// TwinCAT 3 PLC project Untitled1
// ProgramVersion: 3.1.4023.0
// libraries:
//   Tc2_Standard, * (Beckhoff Automation GmbH)
//   Tc2_System, * (Beckhoff Automation GmbH)
//   Tc3_Module, * (Beckhoff Automation GmbH)
// project tree:
//   / PlcTask.TcTTO (not stored)
//   POUs/ MAIN.TcPOU
// real-time tasks:
//   TASK PlcTask: cycle T#10ms, priority 20, ADS port 350
// I/O:
//   DEVICE EtherCAT_Master_EJxxxx, AmsNetId 172.20.30.238.7.1
//     Beckhoff EJ1xxx [EK1100 EtherCAT Coupler (2A E-Bus)]
//       Beckhoff EJ1xxxEK1122 [EK1122 2 port EtherCAT junction]
//         Beckhoff EJ1xxxsub EK1100 [EK1100 EtherCAT Coupler (2A E-Bus)]
//         A_0001(EJ1100-0000-0018) [EJ1100 EtherCAT Coupler (2.2A E-Bus)]
//         A_0002(EJ1101-0022-0016) [EJ1101-0022 EtherCAT Coupler (ID switch)]
//       A_0004(EJ1008-0000-0017) [EJ1008 8Ch. Dig. Input 24V, 3ms]
//       A_0005(EJ1128-0000-0016) [EJ1128 8Ch. Dig. Input 5V / 3.3V DC, 0.05µs]
//       A_0006(EJ1809-0000-0017) [EJ1809 16Ch. Dig. Input 24V, 3ms]
//       A_0007(EJ1819-0000-0017) [EJ1819 16Ch. Dig. Input 24V, 10µs]
//       A_0008(EJ1859-0000-0017) [EJ1859 8Ch. Dig. Input 24V, 3ms, 8Ch. Dig. Output 24V, 0.5A]
//       A_0009(EJ1889-0000-0017) [EJ1889 16Ch. Dig. Input 24V, 3ms, negative]
//       A_0003(EJ1122-0000-0016) [EJ1122 2 port EtherCAT junction]
//     Beckhoff EJ2xxx [EK1100 EtherCAT Coupler (2A E-Bus)]
//       Beckhoff EJ2xxxEK1122 [EK1122 2 port EtherCAT junction]
//         Beckhoff EJ2xxxsub EK1100 [EK1100 EtherCAT Coupler (2A E-Bus)]
//       A_0001(EJ2008-0000-0017) [EJ2008 8Ch. Dig. Output 24V, 0.5A]
//       A_0002(EJ2008-0000-0018) [EJ2008 8Ch. Dig. Output 24V, 0.5A]
//       A_0003(EJ2128-0000-0016) [EJ2128 8Ch. Dig. Output 5V/3.3V, 20mA]
//       A_0004(EJ2502-0000-0023) [EJ2502 2Ch. PWM output, 24V]
//       A_0005(EJ2502-0000-0024) [EJ2502 2Ch. PWM output, 24V]
//       A_0006(EJ2521-0224-0016) [EJ2521-0224 1Ch. Pulse Train 24V DC Output Capture/Compare]
//       A_0007(EJ2522-0000-0022) [EJ2522 2Ch. Pulse Train Output]
//       A_0008(EJ2809-0000-0017) [EJ2809 16Ch. Dig. Output 24V, 0.5A]
//       A_0009(EJ2889-0000-0016) [EJ2889 16Ch. Dig. Output 24V, 0.5A, negative]
//       A_0010(EJ2889-0000-0017) [EJ2889 16Ch. Dig. Output 24V, 0.5A, negative]
//     Beckhoff EJ3xxx [EK1100 EtherCAT Coupler (2A E-Bus)]
//       Beckhoff EJ3xxxEK1122 [EK1122 2 port EtherCAT junction]
//         Beckhoff EJ3xxxsub EK1100 [EK1100 EtherCAT Coupler (2A E-Bus)]
//       A_0001(EJ3004-0000-0019) [EJ3004 4Ch. Ana. Input +/-10V]
//       A_0002(EJ3004-0000-0020) [EJ3004 4Ch. Ana. Input +/-10V]
//       A_0003(EJ3004-0000-0021) [EJ3004 4Ch. Ana. Input +/-10V]
//       A_0004(EJ3048-0000-0020) [EJ3048 8Ch. Ana. Input 0-20mA]
//       A_0005(EJ3058-0000-0020) [EJ3058 8Ch. Ana. Input 4-20mA]
//       A_0006(EJ3068-0000-0020) [EJ3068 8Ch. Ana. Input 0-10V]
//       A_0007(EJ3068-0000-0021) [EJ3068 8Ch. Ana. Input 0-10V]
//       A_0008(EJ3104-0000-0019) [EJ3104 4Ch. Ana. Input +/-10V DIFF]
//       A_0009(EJ3104-0000-0020) [EJ3104 4Ch. Ana. Input +/-10V DIFF]
//       A_0010(EJ3104-0000-0021) [EJ3104 4Ch. Ana. Input +/-10V DIFF]
//       A_0011(EJ3108-0000-0017) [EJ3108 8Ch. Ana. Input +/-10V]
//       A_0012(EJ3108-0000-0018) [EJ3108 8Ch. Ana. Input +/-10V]
//       A_0013(EJ3108-0000-0019) [EJ3108 8Ch. Ana. Input +/-10V]
//       A_0014(EJ3202-0000-0019) [EJ3202 2Ch. Ana. Input PT100 (RTD)]
//       A_0015(EJ3202-0000-0020) [EJ3202 2Ch. Ana. Input PT100 (RTD)]
//       A_0016(EJ3202-0000-0021) [EJ3202 2Ch. Ana. Input PT100 (RTD)]
//       A_0017(EJ3214-0000-0016) [EJ3214 4Ch. Ana. Input PT100 (RTD)]
//       A_0018(EJ3255-0000-0023) [EJ3255 5Ch. potentiometer measurement with sensor supply]
//       A_0019(EJ3318-0000-0017) [EJ3318 8Ch. Ana Input Thermocouple (TC)]
//     Beckhoff EJ4xxx [EK1100 EtherCAT Coupler (2A E-Bus)]
//       Beckhoff EJ4xxxEK1122 [EK1122 2 port EtherCAT junction]
//         Beckhoff EJ4xxxsub EK1100 [EK1100 EtherCAT Coupler (2A E-Bus)]
//       A_0001(EJ4002-0000-0017) [EJ4002 2Ch. Ana. Output 0-10V, 12bit]
//       A_0002(EJ4002-0000-0018) [EJ4002 2Ch. Ana. Output 0-10V, 12bit]
//       A_0003(EJ4004-0000-0020) [EJ4004 4Ch. Ana. Output 0-10V, 12bit]
//       A_0004(EJ4008-0000-0020) [EJ4008 8Ch. Ana. Output 0-10V, 12bit]
//       A_0005(EJ4018-0000-0016) [EJ4018 8Ch. Ana. Output 0-20mA, 12bit]
//       A_0006(EJ4024-0000-0020) [EJ4024 4Ch. Ana. Output 4-20mA, 12bit]
//       A_0007(EJ4132-0000-0019) [EJ4132 2Ch. Ana. Output -10/+10V, 16bit]
//       A_0008(EJ4134-0000-0019) [EJ4134 4Ch. Ana. Output -10/+10V, 16bit]
//       A_0009(EJ4134-0000-0020) [EJ4134 4Ch. Ana. Output -10/+10V, 16bit]
//     Beckhoff EJ5xxx [EK1100 EtherCAT Coupler (2A E-Bus)]
//       Beckhoff EJ5xxxEK1122 [EK1122 2 port EtherCAT junction]
//         Beckhoff EJ5xxxsub EK1100 [EK1100 EtherCAT Coupler (2A E-Bus)]
//       A_0001(EJ5002-0000-0016) [EJ5002 2Ch. SSI Encoder]
//       A_0002(EJ5002-0000-0017) [EJ5002 2Ch. SSI Encoder]
//       A_0003(EJ5101-0000-0016) [EJ5101 1Ch. Inc. Encoder 5V]
//       A_0004(EJ5151-0000-0016) [EJ5151 1Ch. Inc. Encoder]
//     Beckhoff EJ6xxx [EK1100 EtherCAT Coupler (2A E-Bus)]
//       Beckhoff EJ6xxxEK1122 [EK1122 2 port EtherCAT junction]
//         Beckhoff EJ6xxxsub EK1100 [EK1100 EtherCAT Coupler (2A E-Bus)]
//       A_0001(EJ6002-0000-0016) [EJ6002 Interface 2Ch. (RS232/RS485/RS422)]
//       A_0002(EJ6224-0000-0016) [EJ6224 (IO Link Master)]
//         modules: Module 1 (DeviceState Inputs Device), Module 2 (DeviceState Inputs), Module 3 (empty), Module 4 (empty), Module 5 (empty), Module 6 (empty)
//       A_0003(EJ6224-0090-0016) [EJ6224-0090 (IO Link Master, TwinSAFE SC)]
//         modules: Module 1 (DeviceState Inputs Device), Module 2 (DeviceState Inputs), Module 3 (empty), Module 4 (empty), Module 5 (empty), Module 6 (empty)
//     Beckhoff EJ7xxx [EK1100 EtherCAT Coupler (2A E-Bus)]
//       Beckhoff EJ7xxxEK1122 [EK1122 2 port EtherCAT junction]
//         Beckhoff EJ7xxxsub EK1100 [EK1100 EtherCAT Coupler (2A E-Bus)]
//       A_0001(EJ7031-0000-0026) [EJ7031 1Ch. Stepper motor output stage (24V, 1.5A)]
//       A_0002(EJ7037-0000-0020) [EJ7037 1Ch. Stepper motor output stage (24V, 1.5A)]
//       A_0003(EJ7041-0052-0016) [EJ7041-0052 1Ch. Stepper motor output stage (50V, 5A)]
//       A_0004(EJ7047-0000-0018) [EJ7047 1Ch. Stepper motor output stage (50V, 5A)]
//       A_0005(EJ7047-0000-0019) [EJ7047 1Ch. Stepper motor output stage (50V, 5A)]
//       A_0006(EJ7047-0000-0020) [EJ7047 1Ch. Stepper motor output stage (50V, 5A)]
//       A_0007(EJ7342-0000-0019) [EJ7342 2Ch. DC motor output stage (50V, 3.5A)]
//       A_0008(EJ7342-0000-0020) [EJ7342 2Ch. DC motor output stage (50V, 3.5A)]
//       A_0009(EJ7211-0010-0026) [EJ7211-0010 1Ch. MDP742 Servo motor output stage with OCT (50V, 4.5A RMS)]
//       A_0010(EJ7211-0010-0027) [EJ7211-0010 1Ch. MDP742 Servo motor output stage with OCT (50V, 4.5A RMS)]
//       A_0011(EJ7211-0010-0028) [EJ7211-0010 1Ch. MDP742 Servo motor output stage with OCT (50V, 4.5A RMS)]
//       A_0012(EJ7211-0010-0029) [EJ7211-0010 1Ch. MDP742 Servo motor output stage with OCT (50V, 4.5A RMS)]
//       A_0013(EJ7211-0010-0030) [EJ7211-0010 1Ch. MDP742 Servo motor output stage with OCT (50V, 4.5A RMS)]
//       A_0014(EJ7211-0010-0031) [EJ7211-0010 1Ch. MDP742 Servo motor output stage with OCT (50V, 4.5A RMS)]
//       A_0015(EJ7211-0010-0032) [EJ7211-0010 1Ch. MDP742 Servo motor output stage with OCT (50V, 4.5A RMS)]
//       A_0016(EJ7211-0011-0026) [EJ7211-0011 1Ch. DS402 Servo motor output stage with OCT (50V, 4.5A RMS)]
//       A_0017(EJ7211-0011-0027) [EJ7211-0011 1Ch. DS402 Servo motor output stage with OCT (50V, 4.5A RMS)]
//       A_0018(EJ7211-0011-0028) [EJ7211-0011 1Ch. DS402 Servo motor output stage with OCT (50V, 4.5A RMS)]
//       A_0019(EJ7211-0011-0029) [EJ7211-0011 1Ch. DS402 Servo motor output stage with OCT (50V, 4.5A RMS)]
//       A_0020(EJ7211-0011-0030) [EJ7211-0011 1Ch. DS402 Servo motor output stage with OCT (50V, 4.5A RMS)]
//       A_0021(EJ7211-0011-0031) [EJ7211-0011 1Ch. DS402 Servo motor output stage with OCT (50V, 4.5A RMS)]
//       A_0022(EJ7211-0011-0032) [EJ7211-0011 1Ch. DS402 Servo motor output stage with OCT (50V, 4.5A RMS)]
//       A_0023(EJ7211-9414-0029) [EJ7211-9414 1Ch. MDP742 Servo motor output stage with OCT (50V, 4.5A RMS) , TwinSAFE SC]
//       A_0024(EJ7211-9414-0030) [EJ7211-9414 1Ch. MDP742 Servo motor output stage with OCT (50V, 4.5A RMS) , TwinSAFE SC]
//       A_0025(EJ7211-9414-0031) [EJ7211-9414 1Ch. MDP742 Servo motor output stage with OCT (50V, 4.5A RMS) , TwinSAFE SC]
//       A_0026(EJ7211-9414-0032) [EJ7211-9414 1Ch. MDP742 Servo motor output stage with OCT (50V, 4.5A RMS) , TwinSAFE SC]
//       A_0027(EJ7211-9415-0029) [EJ7211-9415 1Ch. DS402 Servo motor output stage with OCT (50V, 4.5A RMS), TwinSAFE SC]
//       A_0028(EJ7211-9415-0030) [EJ7211-9415 1Ch. DS402 Servo motor output stage with OCT (50V, 4.5A RMS), TwinSAFE SC]
//       A_0029(EJ7211-9415-0031) [EJ7211-9415 1Ch. DS402 Servo motor output stage with OCT (50V, 4.5A RMS), TwinSAFE SC]
//       A_0030(EJ7211-9415-0032) [EJ7211-9415 1Ch. DS402 Servo motor output stage with OCT (50V, 4.5A RMS), TwinSAFE SC]
//       A_0031(EJ7334-0008-0016) [EJ7334-0008 4 Ch. Bi-/8 Ch. Unidirectional DC motor output stage (24 V, 8 A overall current)]
//       A_0032(EJ7411-0000-0018) [EJ7411 BLDC Terminal with incremental encoder/Hall, 50 V DC, 4.5 A]
//     Beckhoff EJ9xxx [EK1100 EtherCAT Coupler (2A E-Bus)]
//       Beckhoff EJ9xxxEK1122 [EK1122 2 port EtherCAT junction]
//         Beckhoff EJ9xxxsub EK1100 [EK1100 EtherCAT Coupler (2A E-Bus)]
//       A_0001(EJ9001-0000-0016) [EJ9001 placeholder module]
//       A_0002(EJ9505-0000-0016) [EJ9505 Power supply module 5V]
//       A_0003(EJ9576-0000-0018) [EJ9576 Brake chopper terminal]
//       A_0004(EJ9576-0000-0019) [EJ9576 Brake chopper terminal]
//       A_0005(EJ9576-0000-0020) [EJ9576 Brake chopper terminal]
//       A_0006(EJ9576-0000-0022) [EJ9576 Brake chopper terminal]
//       A_0007 (EJ9400-0000) [EJ9400-0000 Power supply module 2,5A]
//       A_0008 (EJ9404-0000) [EJ9404-0000 Power supply module 12A]
//     Beckhoff EJx9xx [EK1100 EtherCAT Coupler (2A E-Bus)]
//       Beckhoff EJx9xxEK1122 [EK1122 2 port EtherCAT junction]
//         Beckhoff EJx9xxsub EK1100 [EK1100 EtherCAT Coupler (2A E-Bus)]
//       A_0001(EJ1914-0000-0017) [EJ1914-0000-0017]
//         modules: Module 1 (FSOE), Module 2 (DEVICEIO), Module 3 (FSLOGIC)
//       A_0002(EJ1914-0000-0018) [EJ1914, 4Ch. Safety Input 24V, TwinSAFE]
//         modules: Module 1 (FSOE), Module 2 (DEVICEIO), Module 3 (FSLOGIC)
//       A_0003(EJ1918-0000-0017) [EJ1918-0000-0017]
//         modules: Module 1 (FSOE), Module 2 (DEVICEIO), Module 3 (FSLOGIC)
//       A_0004(EJ1918-0000-0018) [EJ1918, 8Ch. Safety Input 24V, TwinSAFE]
//         modules: Module 1 (FSOE), Module 2 (DEVICEIO), Module 3 (FSLOGIC)
//       A_0005(EJ1957-0000-0017) [EJ1957-0000-0017]
//         modules: Module 1 (FSOE), Module 2 (FSOUT), Module 3 (DEVICEIO), Module 4 (FSLOGIC)
//       A_0006(EJ1957-0000-0018) [EJ1957, 8Ch. Safety Input 24V, 4Ch. Safety Output 24V, 0.5A, TwinSAFE]
//         modules: Module 1 (FSOE), Module 2 (FSOUT), Module 3 (DEVICEIO), Module 4 (FSLOGIC)
//       A_0007(EJ2914-0000-0017) [EJ2914-0000-0017]
//         modules: Module 1 (FSOE), Module 2 (FSOUT), Module 3 (DEVICEIO), Module 4 (FSLOGIC)
//       A_0008(EJ2914-0000-0018) [EJ2914, 4Ch. Safety Output 24V, 0.5A, TwinSAFE]
//         modules: Module 1 (FSOE), Module 2 (FSOUT), Module 3 (DEVICEIO), Module 4 (FSLOGIC)
//       A_0009(EJ2918-0000-0017) [EJ2918-0000-0017]
//         modules: Module 1 (FSOE), Module 2 (FSOUT), Module 3 (DEVICEIO), Module 4 (FSLOGIC)
//       A_0010(EJ2918-0000-0018) [EJ2918, 8Ch. Safety Output 24V, 0.5A, TwinSAFE]
//         modules: Module 1 (FSOE), Module 2 (FSOUT), Module 3 (DEVICEIO), Module 4 (FSLOGIC)
//       A_0011(EJ6910-0000-0018) [EJ6910, TwinSAFE PLC]
//       A_0012(EJ6910-0000-0020) [EJ6910, TwinSAFE PLC]
//   DEVICE EtherCAT_Master_EKxxxx, AmsNetId 172.20.30.238.8.1
//     Beckhoff EK11xx [EK1100 EtherCAT Coupler (2A E-Bus)]
//       Beckhoff EK11xxEK1122 [EK1122 2 port EtherCAT junction]
//         Beckhoff EK11xxsub EK1100 [EK1100 EtherCAT Coupler (2A E-Bus)]
//         A_0001(EK1100-0000-0000) [EK1100 EtherCAT Coupler (0.5A E-Bus)]
//         A_0002(EK1100-0000-0001) [EK1100 EtherCAT Coupler (2A E-Bus)]
//         A_0003(EK1100-0000-0016) [EK1100 EtherCAT Coupler (2A E-Bus)]
//         A_0004(EK1100-0000-0017) [EK1100 EtherCAT Coupler (2A E-Bus)]
//         A_0005(EK1100-0000-0018) [EK1100 EtherCAT Coupler (2A E-Bus)]
//         A_0006(EK1100-0008-0016) [EK1100-0008 EtherCAT Coupler M8 (2A E-Bus)]
//         A_0009(EK1101-0000-0016) [EK1101 EtherCAT Coupler (2A E-Bus, ID switch)]
//         A_0010(EK1101-0000-0017) [EK1101 EtherCAT Coupler (2A E-Bus, ID switch)]
//         A_0011(EK1101-0000-0018) [EK1101 EtherCAT Coupler (2A E-Bus, ID switch)]
//         A_0012(EK1101-0008-0016) [EK1101-0008 EtherCAT Coupler M8 (2A E-Bus, ID switch)]
//         A_0013(EK1101-0010-0016) [EK1101-0010 EtherCAT Coupler (2A E-Bus, ID switch, Extended Distance)]
//         A_0008(EK1100-0030-0017) [EK1100-0030 EtherCAT Coupler (2A E-Bus, 4kV galv. iso.)]
//         A_0007(EK1100-0030-0016) [EK1100-0030 EtherCAT Coupler (2A E-Bus, 4kV galv. iso.)]
//       A_0018(EK1110-0043-0016) [EK1110-0043 EtherCAT EJ coupler]
//       A_0024(EK1122-0008-0016) [EK1122-0008 2 port EtherCAT junction M8]
//       A_0023(EK1122-0000-0018) [EK1122 2 port EtherCAT junction]
//       A_0022(EK1122-0000-0017) [EK1122 2 port EtherCAT junction]
//       A_0021(EK1122-0000-0016) [EK1122 2 port EtherCAT junction]
//       A_0020(EK1121-0010-0016) [EK1121-0010 1 port EtherCAT junction (Extended Distance)]
//       A_0019(EK1110-0044-0016) [EK1110-0044 EtherCAT EJ coupler]
//       A_0017(EK1110-0008-0016) [EK1110-0008 EtherCAT extension M8]
//       A_0016(EK1110-0000-0017) [EK1110 EtherCAT extension]
//       A_0015(EK1110-0000-0016) [EK1110 EtherCAT extension]
//       A_0014(EK1110-0000-0000) [EK1110 EtherCAT extension]
//     Beckhoff EK12xx [EK1100 EtherCAT Coupler (2A E-Bus)]
//       Beckhoff EK12xxEK1122 [EK1122 2 port EtherCAT junction]
//         Beckhoff EK12xxsub EK1100 [EK1100 EtherCAT Coupler (2A E-Bus)]
//         A_0002(EK1200-7000-0000) [EK1200-7000 EtherCAT Power supply (1,5A E-Bus)]
//         A_0001(EK1200-5000-0000) [EK1200-5000 EtherCAT Power supply (2A E-Bus)]
//     Beckhoff EK13xx [EK1100 EtherCAT Coupler (2A E-Bus)]
//       Beckhoff EK13xxEK1122 [EK1122 2 port EtherCAT junction]
//         Beckhoff EK13xxsub EK1100 [EK1100 EtherCAT Coupler (2A E-Bus)]
//         A_0001(EK1300-0000-0017) [EK1300 EtherCAT P Coupler (2A E-Bus)]
//       A_0003(EK1322-0000-0017) [EK1322 2-port EtherCAT P junction with feed-in]
//       A_0002(EK1310-0000-0017) [EK1310 EtherCAT P extension with feed-in]
//     Beckhoff EK15xx [EK1100 EtherCAT Coupler (2A E-Bus)]
//       Beckhoff EK15xxEK1122 [EK1122 2 port EtherCAT junction]
//         Beckhoff EK15xxsub EK1100 [EK1100 EtherCAT Coupler (2A E-Bus)]
//         A_0001(EK1501-0000-0016) [EK1501 EtherCAT Coupler (2A E-Bus, FX-MultiMode, ID switch)]
//         A_0002(EK1501-0000-0017) [EK1501 EtherCAT Coupler (2A E-Bus, FX-MultiMode, ID switch)]
//         A_0003(EK1501-0000-0018) [EK1501 EtherCAT Coupler (2A E-Bus, FX-MultiMode, ID switch)]
//         A_0004(EK1501-0000-0019) [EK1501 EtherCAT Coupler (2A E-Bus, FX-MultiMode, ID switch)]
//         A_0005(EK1501-0010-0016) [EK1501-0010 EtherCAT Coupler (2A E-Bus, FX-SingleMode, ID switch)]
//         A_0006(EK1501-0010-0017) [EK1501-0010 EtherCAT Coupler (2A E-Bus, FX-SingleMode, ID switch)]
//         A_0007(EK1501-0010-0018) [EK1501-0010 EtherCAT Coupler (2A E-Bus, FX-SingleMode, ID switch)]
//         A_0008(EK1501-0100-0016) [EK1501-0100 EtherCAT Coupler (2A E-Bus, FX-MultiMode, media converter, ID switch)]
//         A_0020(EK1541-0000-0016) [EK1541 EtherCAT Coupler (2A E-Bus, POF, ID switch)]
//         A_0021(EK1541-0000-0017) [EK1541 EtherCAT Coupler (2A E-Bus, POF, ID switch)]
//         A_0022(EK1541-0000-0018) [EK1541 EtherCAT Coupler (2A E-Bus, POF, ID switch)]
//       A_0025(EK1561-0000-0018) [EK1561 1 port EtherCAT junction (POF)]
//       A_0024(EK1561-0000-0017) [EK1561 1 port EtherCAT junction (POF)]
//       A_0023(EK1561-0000-0016) [EK1561 1 port EtherCAT junction (POF)]
//       A_0019(EK1521-0010-0020) [EK1521-0010 1 port EtherCAT junction (FX-SingleMode)]
//       A_0018(EK1521-0010-0019) [EK1521-0010 1 port EtherCAT junction (FX-SingleMode)]
//       A_0017(EK1521-0010-0018) [EK1521-0010 1 port EtherCAT junction (FX-SingleMode)]
//       A_0016(EK1521-0010-0017) [EK1521-0010 1 port EtherCAT junction (FX-SingleMode)]
//       A_0015(EK1521-0010-0016) [EK1521-0010 1 port EtherCAT junction (FX-SingleMode)]
//       A_0014(EK1521-0000-0021) [EK1521 1 port EtherCAT junction (FX-MultiMode)]
//       A_0013(EK1521-0000-0020) [EK1521 1 port EtherCAT junction (FX-MultiMode)]
//       A_0012(EK1521-0000-0019) [EK1521 1 port EtherCAT junction (FX-MultiMode)]
//       A_0011(EK1521-0000-0018) [EK1521 1 port EtherCAT junction (FX-MultiMode)]
//       A_0010(EK1521-0000-0017) [EK1521 1 port EtherCAT junction (FX-MultiMode)]
//       A_0009(EK1521-0000-0016) [EK1521 1 port EtherCAT junction (FX-MultiMode)]
//     Beckhoff EK18xx [EK1100 EtherCAT Coupler (2A E-Bus)]
//       Beckhoff EK18xxEK1122 [EK1122 2 port EtherCAT junction]
//         Beckhoff EK18xxsub EK1100 [EK1100 EtherCAT Coupler (2A E-Bus)]
//         A_0001(EK1814-0000-0016) [EK1814 EtherCAT IO-Coupler  (0,5A E-Bus, 4 Ch. Dig. In, 3ms, 4 Ch. Dig. Out 24V, 0,5A)]
//         A_0002(EK1814-0000-0017) [EK1814 EtherCAT IO-Coupler  (1A E-Bus, 4 Ch. Dig. In, 3ms, 4 Ch. Dig. Out 24V, 0,5A)]
//         A_0003(EK1814-0000-0018) [EK1814 EtherCAT IO-Coupler  (1A E-Bus, 4 Ch. Dig. In, 3ms, 4 Ch. Dig. Out 24V, 0,5A)]
//         A_0004(EK1814-0000-0019) [EK1814 EtherCAT IO-Coupler  (1A E-Bus, 4 Ch. Dig. In, 3ms, 4 Ch. Dig. Out 24V, 0,5A)]
//         A_0005(EK1818-0000-0016) [EK1818 EtherCAT IO-Coupler  (1A E-Bus, 8 Ch. Dig. In, 3ms, 4 Ch. Dig. Out 24V, 0,5A)]
//         A_0006(EK1818-0000-0017) [EK1818 EtherCAT IO-Coupler  (1A E-Bus, 8 Ch. Dig. In, 3ms, 4 Ch. Dig. Out 24V, 0,5A)]
//         A_0007(EK1818-0000-0018) [EK1818 EtherCAT IO-Coupler  (1A E-Bus, 8 Ch. Dig. In, 3ms, 4 Ch. Dig. Out 24V, 0,5A)]
//         A_0008(EK1828-0000-0016) [EK1828 EtherCAT IO-Coupler  (1A E-Bus, 4 Ch. Dig. In, 3ms, 8 Ch. Dig. Out 24V, 0,5A)]
//         A_0009(EK1828-0000-0017) [EK1828 EtherCAT IO-Coupler  (1A E-Bus, 4 Ch. Dig. In, 3ms, 8 Ch. Dig. Out 24V, 0,5A)]
//         A_0010(EK1828-0000-0018) [EK1828 EtherCAT IO-Coupler  (1A E-Bus, 4 Ch. Dig. In, 3ms, 8 Ch. Dig. Out 24V, 0,5A)]
//         A_0011(EK1828-0010-0016) [EK1828-0010 EtherCAT IO-Coupler  (1A E-Bus, 8 Ch. Dig. Out 24V, 0,5A)]
//         A_0012(EK1828-0010-0017) [EK1828-0010 EtherCAT IO-Coupler  (1A E-Bus, 8 Ch. Dig. Out 24V, 0,5A)]
//         A_0013(EK1828-0010-0018) [EK1828-0010 EtherCAT IO-Coupler  (1A E-Bus, 8 Ch. Dig. Out 24V, 0,5A)]
//     Beckhoff EKM1xxx [EK1100 EtherCAT Coupler (2A E-Bus)]
//       Beckhoff EKM1xxxEK1122 [EK1122 2 port EtherCAT junction]
//         Beckhoff EKM1xxxsub EK1100 [EK1100 EtherCAT Coupler (2A E-Bus)]
//         A_0001(EKM1101-0000-0016) [EKM1101 EtherCAT Coupler  (2A E-Bus, ID switch, Diagnostics, isolated)]
//         A_0002(EKM1101-0000-0017) [EKM1101 EtherCAT Coupler  (2A E-Bus, ID switch, Diagnostics, isolated)]
//         A_0003(EKM1101-0000-0018) [EKM1101 EtherCAT Coupler  (2A E-Bus, ID switch, Diagnostics, isolated)]
//         A_0004(EKM1101-0000-0019) [EKM1101 EtherCAT Coupler  (2A E-Bus, ID switch, Diagnostics, isolated)]
//         A_0005(EKM1101-0000-0020) [EKM1101 EtherCAT Coupler  (2A E-Bus, ID switch, Diagnostics, isolated)]
//     Beckhoff EKx9xx [EK1100 EtherCAT Coupler (2A E-Bus)]
//       Beckhoff EKx9xxEK1122 [EK1122 2 port EtherCAT junction]
//         Beckhoff EKx9xxsub EK1100 [EK1100 EtherCAT Coupler (2A E-Bus)]
//         A_0001(EK1960-0000-0019) [EK1960-0000 TwinSAFE-Compact-Controller (RJ45)]
//           modules: Module 1 (FSoE), Module 2 (FSOUT), Module 3 (FSLOGIC)
//         A_0002(EK1960-0000-0021) [EK1960-0000 TwinSAFE-Compact-Controller (RJ45)]
//           modules: Module 1 (FSoE), Module 2 (FSOUT), Module 3 (FSLOGIC)
//         A_0003(EK1960-0008-0019) [EK1960-0008 TwinSAFE-Compact-Controller (M8)]
//           modules: Module 1 (FSoE), Module 2 (FSOUT), Module 3 (FSLOGIC)
//         A_0004(EK1960-0008-0021) [EK1960-0008 TwinSAFE-Compact-Controller (M8)]
//           modules: Module 1 (FSoE), Module 2 (FSOUT), Module 3 (FSLOGIC)
//         A_0005(EK1960-2600-0019) [EK1960-2600 TwinSAFE-Compact-Controller (4 x Relay, RJ45)]
//           modules: Module 1 (FSoE), Module 2 (FSOUT), Module 3 (FSLOGIC)
//         A_0006(EK1960-2600-0021) [EK1960-2600 TwinSAFE-Compact-Controller (4 x Relay, RJ45)]
//           modules: Module 1 (FSoE), Module 2 (FSOUT), Module 3 (FSLOGIC)
//         A_0007(EK1960-2608-0019) [EK1960-2608 TwinSAFE-Compact-Controller (4 x Relay, M8)]
//           modules: Module 1 (FSoE), Module 2 (FSOUT), Module 3 (FSLOGIC)
//         A_0008(EK1960-2608-0021) [EK1960-2608 TwinSAFE-Compact-Controller (4 x Relay, M8)]
//           modules: Module 1 (FSoE), Module 2 (FSOUT), Module 3 (FSLOGIC)
//     Beckhoff EKxxxx-0080 [EK1100 EtherCAT Coupler (2A E-Bus)]
//       Beckhoff EKxxxx-0080EK1122 [EK1122 2 port EtherCAT junction]
//         Beckhoff EKxxxx-0080sub EK1100 [EK1100 EtherCAT Coupler (2A E-Bus)]
//       A_0006(EK1122-0080-0019) [EK1122-0080 2 port EtherCAT junction (Fast Hot Connect)]
//       A_0005(EK1122-0080-0018) [EK1122-0080 2 port EtherCAT junction (Fast Hot Connect)]
//       A_0004(EK1122-0080-0017) [EK1122-0080 2 port EtherCAT junction (Fast Hot Connect)]

// ---- POUs/MAIN.TcPOU
PROGRAM MAIN
VAR
END_VAR

END_PROGRAM
